PROGRAM PRG_PING_DMX
  VAR
    udiPingTime : UDINT;
    udiDMXnodeReachable : UDINT;
    udiPreviousReachable : UDINT := 16#FFFFFFFF;  (* Last reported result, so the log fires on transitions only. The sentinel differs from every SysSockPing return, so the first pass still logs. *)
    sBrokerHost : STRING;  (* The broker's host without its port. GVL_MQTT.broker carries host:port and SysSockPing wants the host on its own, so it is split here rather than duplicated as a second constant that would drift. Assumes an address of the form ip:port, which is what GVL_MQTT.broker has always held. *)
    iColon : INT;
    udiBrokerPingTime : UDINT;
    udiBrokerReachable : UDINT;
    bPreviousBrokerReachable : BOOL := FALSE;  (* Last logged verdict, so the log fires on transitions only. Deliberately initialised FALSE where bBrokerReachable starts TRUE, so the first verdict is logged whichever way it goes. *)
    uiBrokerPingFails : UINT;  (* Consecutive failed broker pings. One lost ICMP packet must not turn a cabinet LED red, and SysSockPing returns codes that are neither 0 nor 5 - the DMX ping above has always ignored those rather than acting on them. Counting instead of enumerating return codes means an unknown code is treated as a failure without a single one of them being able to flip the light. *)
  END_VAR
  VAR CONSTANT
    cuiBrokerPingFailsForRed : UINT := 2;  (* Failed pings in a row before the broker counts as unreachable. Two, against a 10 s task, means U1 goes red within about 20 s of the cable coming out and green again within 10 s of it going back in. Lower the Ping task period if that is not quick enough; do not lower this to one. *)
  END_VAR

                    (* Ping the DMX artNet node *)
udiDMXnodeReachable := SysSockPing(szIPAddress:=GVL_DMX.IP, ulTimeout:=100, pulReplyTime:= ADR(udiPingTime));

IF udiDMXnodeReachable = 0 THEN
    PFC.SetLed(which:=PFC.LED.U3, how:=PFC.LedState.STATIC_GRN);
	IF udiDMXnodeReachable <> udiPreviousReachable THEN
		GVL_MQTT.PLC_Device.SendLogMessage('DMX ping OK');
	END_IF
ELSIF udiDMXnodeReachable = 5 THEN
     PFC.SetLed(which:=PFC.LED.U3, how:=PFC.LedState.BLINK_RED);
	IF udiDMXnodeReachable <> udiPreviousReachable THEN
		GVL_MQTT.PLC_Device.SendLogMessage('DMX ping Error');
	END_IF
END_IF

udiPreviousReachable := udiDMXnodeReachable;

(* Ping the MQTT broker as well, because U1 needs something the MQTT client cannot
   tell it. MQTT_CONNECTED does not notice a pulled network cable: a TCP socket with
   nothing to report stays open until a retransmit finally gives up, which is minutes
   rather than seconds, so the client goes on believing it has a session. Verified on
   the bench - LAN cable out, MQTT_CONNECTED still TRUE, U1 still green. ICMP notices
   in one task cycle, and the debounce below spends one more, so U1 turns red within
   about 20 s of the cable coming out and green within 10 s of it going back in.

   PRG_MQTT owns the LED; this only reports what it found. *)
iColon := FIND(GVL_MQTT.broker, ':');
IF iColon > 1 THEN
	sBrokerHost := LEFT(GVL_MQTT.broker, iColon - 1);
ELSE
	(* No port in the address, so it is already just the host. FIND returns 0 when
	   it matches nothing, which this also covers. *)
	sBrokerHost := GVL_MQTT.broker;
END_IF

udiBrokerReachable := SysSockPing(szIPAddress := sBrokerHost, ulTimeout := 100,
	pulReplyTime := ADR(udiBrokerPingTime));

(* Debounced, because one lost packet is not an outage. A success clears the count
   immediately, so recovery is as fast as the task; failures have to stack up. *)
IF udiBrokerReachable = 0 THEN
	uiBrokerPingFails := 0;
ELSIF uiBrokerPingFails < cuiBrokerPingFailsForRed THEN
	uiBrokerPingFails := uiBrokerPingFails + 1;
END_IF

GVL_MQTT.bBrokerReachable := (uiBrokerPingFails < cuiBrokerPingFailsForRed);

(* Log the debounced verdict, not the raw return code - otherwise a run of odd
   codes would log on every one of them. *)
IF GVL_MQTT.bBrokerReachable <> bPreviousBrokerReachable THEN
	IF GVL_MQTT.bBrokerReachable THEN
		GVL_MQTT.PLC_Device.SendLogMessage('MQTT broker ping OK');
	ELSE
		(* This one cannot be delivered while the broker is away; it queues and
		   arrives on reconnect, which is what makes the outage visible after the
		   fact rather than not at all. *)
		GVL_MQTT.PLC_Device.SendLogMessage('MQTT broker ping Error');
	END_IF
	bPreviousBrokerReachable := GVL_MQTT.bBrokerReachable;
END_IF

                  
END_PROGRAM

PROGRAM PRG_DALI_VERIFY
  VAR
    Ballast : WagoAppDALI.typBallast := (bAddress := 0, xIsGroup := FALSE, bPortDALI := 1);  (* A ballast on the first 753-647 of this device, short address 0. The values are arbitrary: nothing here is downloaded. What matters is that every type and every call in the DALI chain is compiled on every build. *)
    fbDaliMaster : WagoAppDALI.FbDaliMaster;  (* The master, and the block under test. *)
    fbDimmer : FB_OUTPUT_DIMMER_DALI_MQTT;
  END_VAR

                    // Run the master before anything else, bound to the 753-647 on this device's own
// K-bus. This binding is the whole point of the second controller: I_Port wants a
// WagoTypesModule_753_647.I_Port_753_647, which only WAGO's device description
// creates, and that description does not fit the G1 lab device's bus.
fbDaliMaster(
	bPortDALI := 1,
	I_Port := IoConfig_Globals.DALI_753_647);

// The block under test. No InitMqtt and no InitMqttDiscovery: this application
// never runs, and calling them would only invent a Home Assistant entity for a
// controller that does not exist.
fbDimmer(
	BALLAST := Ballast,
	TOGGLE := FALSE,
	P_LONG := FALSE);

                  
END_PROGRAM

CONFIGURATION Wago_PFC200_G1_Lab
  RESOURCE HomeAutomation ON PLC
    {attribute 'qualified_only'}
    VAR_GLOBAL CONSTANT  (* GVL_MQTT *)
      MQTT_TOPIC_LEN : INT := 160;  (* Widths for topics and topic fragments. These used to be spelled out at five different values for the same conceptual string, and IEC string assignment and CONCAT both truncate without any error - so every mismatch was a silent failure point. The tightest real chain: a 28-character prefix like 'Devices/PLC/Lab/Out/Dimmers/' plus a 40-character instance name plus '/OUT' already reached the old STRING(100) limit, after which Home Assistant sees a truncated state topic and the entity goes quietly unavailable. *)
      MQTT_SUFFIX_LEN : INT := 64;
      clientID : STRING := 'PLC-Lab';  (* Broker setup *)
      broker : STRING := '10.101.1.11:1883';
      fbMqttPublishQueue : FB_MQTT_PUBLISH_QUEUE;  (* use the below for username password authentication to broker broker :STRING:='user:password@192.168.1.36:1883'; Shared Variables for MQTT publish communication *)
      collector_FB_OUTPUT_SWITCH_MQTT : MQTT.CallbackCollector;  (* Shared Variables for MQTT subscribe communication *)
      collector_FB_OUTPUT_COVER_MQTT : MQTT.CallbackCollector;
      collector_FB_DIMMER_MQTT : MQTT.CallbackCollector;
      collector_FB_RS485_MQTT : MQTT.CallbackCollector;
      collector_FB_HVAC_MQTT : MQTT.CallbackCollector;
      MQTT_QOS_EXACTLY_ONCE : MQTT.QoS := MQTT.QoS.ExactlyOnce;  (* QOS Constants *)
      MqttMain : STRING(16) := 'Devices/';  (* Topics *)
      MqttType : STRING(16) := 'PLC/';
      MqttDevice : STRING(16) := 'Lab/';
      MqttBaseTopic : STRING(GVL_MQTT.MQTT_TOPIC_LEN) := 'CONCAT(CONCAT(MqttMain, MqttType), MqttDevice)';  (* e.g. Devices/PLC/House *)
      MqttDiagnosticTopic : STRING(GVL_MQTT.MQTT_TOPIC_LEN) := 'CONCAT(MqttBaseTopic, 'diagnostic')';
      MqttAvailabilityTopic : STRING(GVL_MQTT.MQTT_TOPIC_LEN) := 'CONCAT(MqttBaseTopic, 'availability')';
      MqttAvailabilityOnlinePayload : STRING(20) := 'online';
      MqttAvailabilityOfflinePayload : STRING(20) := 'offline';
      MQTTAvailabilityHartbeatTime : TIME := TIME#5s0ms;
      MqttHADiscoveryPrefix : STRING(16) := 'homeassistant/';
      PLC_Device : FB_PLC_MQTT_DISCOVERY_DEVICE;  (* HOME ASSISTANT DISCOVERY VIA MQTT *)
      OWD_MULTISENSOR_01 : FB_1WIRE_MQTT_DISCOVERY_DEVICE;
      MqttPushbuttonPrefix : STRING(GVL_MQTT.MQTT_TOPIC_LEN) := 'CONCAT(MqttBaseTopic, 'Out/DigitalInputs/Pushbuttons/')';  (* FB Topics *)
      MqttPubSwitchPrefix : STRING(GVL_MQTT.MQTT_TOPIC_LEN) := 'CONCAT(MqttBaseTopic, 'Out/DigitalOutputs/')';
      MqttSubSwitchPrefix : STRING(GVL_MQTT.MQTT_TOPIC_LEN) := 'CONCAT(MqttBaseTopic, 'In/DigitalOutputs/')';
      MqttPubCoverPrefix : STRING(GVL_MQTT.MQTT_TOPIC_LEN) := 'CONCAT(MqttBaseTopic, 'Out/Covers/')';
      MqttSubCoverPrefix : STRING(GVL_MQTT.MQTT_TOPIC_LEN) := 'CONCAT(MqttBaseTopic, 'In/Covers/')';
      MqttPubDimmerPrefix : STRING(GVL_MQTT.MQTT_TOPIC_LEN) := 'CONCAT(MqttBaseTopic, 'Out/Dimmers/')';
      MqttSubDimmerPrefix : STRING(GVL_MQTT.MQTT_TOPIC_LEN) := 'CONCAT(MqttBaseTopic, 'In/Dimmers/')';
      MqttPubRS485Prefix : STRING(GVL_MQTT.MQTT_TOPIC_LEN) := 'CONCAT(MqttBaseTopic, 'Out/RS485/')';
      MqttSubRS485Prefix : STRING(GVL_MQTT.MQTT_TOPIC_LEN) := 'CONCAT(MqttBaseTopic, 'In/RS485/')';
      MqttPubHVACPrefix : STRING(GVL_MQTT.MQTT_TOPIC_LEN) := 'CONCAT(MqttBaseTopic, 'Out/HVAC/')';
      MqttPubAnalogInputPrefix : STRING(GVL_MQTT.MQTT_TOPIC_LEN) := 'CONCAT(MqttBaseTopic, 'Out/AnalogInputs/')';  (* On-board analog inputs: an RTD channel on a 750-463, and anything else measured by the PLC itself rather than over a bus. Publish only - there is nothing to command on an input. *)
      MqttSubHVACPrefix : STRING(GVL_MQTT.MQTT_TOPIC_LEN) := 'CONCAT(MqttBaseTopic, 'In/HVAC/')';
      MqttSubSwitchTopic : STRING(GVL_MQTT.MQTT_TOPIC_LEN) := 'CONCAT(MqttSubSwitchPrefix, '+')';  (* Wildcard subscriptions *)
      MqttSubCoverTopic : STRING(GVL_MQTT.MQTT_TOPIC_LEN) := 'CONCAT(MqttSubCoverPrefix, '#')';  (* '#', not '+': the position command topic sits one level below the cover's own topic - .../In/Covers/FB_X/POSITION - and a single-level wildcard would not deliver it. The older cover block's topics still match. *)
      MqttSubDimmerTopic : STRING(GVL_MQTT.MQTT_TOPIC_LEN) := 'CONCAT(MqttSubDimmerPrefix, '#')';
      MqttSubRS485Topic : STRING(GVL_MQTT.MQTT_TOPIC_LEN) := 'CONCAT(MqttSubRS485Prefix, '#')';
      MqttSubHVACTopic : STRING(GVL_MQTT.MQTT_TOPIC_LEN) := 'CONCAT(MqttSubHVACPrefix, '#')';
      bBrokerReachable : BOOL := TRUE;  (* TRUE while the broker host answers an ICMP ping. Written by PRG_PING_DMX, read by PRG_MQTT, which ANDs it with the client's own MQTT_CONNECTED before deciding what U1 shows. It is not redundant. MQTT_CONNECTED does not notice a pulled network cable: TCP has nothing to report until a retransmit gives up, so the client can hold a dead socket open for minutes. Measured on the bench - cable out, U1 stayed green. ICMP notices within one cycle of the Ping task. Starts TRUE so it means 'not known to be unreachable': until the Ping task has an opinion, U1 follows MQTT_CONNECTED alone rather than blinking red through a healthy startup. *)
      MQTT_LANE_MAIN : INT := 0;
      MQTT_LANE_RS485 : INT := 1;
      MQTT_LANE_HVAC : INT := 2;
      tMqttReconnectRestMin : TIME := TIME#1s0ms;  (* Reconnect pacing, read by PRG_MQTT. They live here rather than in an FB_init argument or an initialiser because both of those are stored outside the declaration text, where a scripted edit cannot reach them. First pause after a session drops, and the ceiling the pause doubles towards. One second is short enough that an ordinary reconnect is not noticeably slower; a minute is the worst the broker ever sees. *)
      tMqttReconnectRestMax : TIME := TIME#1m0s0ms;
      tMqttSessionStable : TIME := TIME#30s0ms;  (* How long a session has to last before it counts as a real one. Long enough that a session which dies on arrival cannot clear the backoff, short enough that a healthy reconnect clears it well before the next heartbeat. *)
      tMqttStall : TIME := TIME#5m0s0ms;  (* No stable session for this long is a stall, not bad luck: the client stops trying for tMqttStallCoolDown and then starts again. *)
      tMqttStallCoolDown : TIME := TIME#1m0s0ms;
    END_VAR
    {attribute 'qualified_only'}
    VAR_GLOBAL  (* GVL_DMX *)
      IP : STRING := '10.1.1.4';  (* unicast: 10.1.1.4 multicast: 10.1.1.255 broadcast: 255.255.255.255 *)
      DMX : oscat_network.NETWORK_BUFFER_SHORT;
    END_VAR
    {attribute 'qualified_only'}
    VAR_GLOBAL  (* GVL_RS485 *)
      FB_RS485_EASTRON_SDM220_1 : FB_RS485_EASTRON_SDM220_MQTT := (FriendlyName := 'Lab PLC SDM220 energy meter');  (* RS485 *)
      FB_RS485_DUCO_DUCOBOX_HOME : FB_RS485_DUCO_DUCOBOX_FOCUS_MQTT;
      FB_RS485_1WIRE_MULTISENSOR_01 : FB_RS485_ESERA_OWD_MQTT;
      FB_RS485_EASTRON_SDM630_1 : FB_RS485_EASTRON_SDM630_MQTT := (FriendlyName := 'Lab PLC energy meter');  (* Self-wiring: FriendlyName is what turns the MQTT and discovery wiring on, so this needs no Init call in RS485_INIT - only registration on the bus. *)
      FB_RS485_EASTRON_SDM_POWER_1 : FB_RS485_EASTRON_SDM_POWER_MQTT := (FriendlyName := 'Lab PLC SDM power meter');  (* Registered on the bus and pointed at the SAME meter as FB_RS485_EASTRON_SDM220_1 above (Modbus address 1), declared as an SDM220. That is deliberate on two counts. It is the only call site this block has, and an unreferenced POU is never compiled - without an instance somewhere in the application a broken edit to it would pass verify with a clean build. And because both blocks decode active power out of the same register (30013), the two publish the same number continuously: a persistent difference between .../FB_RS485_EASTRON_SDM_POWER_1/ACTP and .../FB_RS485_EASTRON_SDM220_1/ACTP means one of them has stopped decoding correctly. There is no SDM120 or SDM630 here, so this is the only way the block is exercised at all. *)
      FB_RS485_SEN0492_1 : FB_RS485_DFROBOT_SEN0492_MQTT := (FriendlyName := 'Lab PLC rangefinder');  (* DFRobot SEN0492 laser rangefinder, 4 cm to 4 m over RS485. Left at its factory slave address 16#50, which collides with nothing on this bus - the Eastron meters sit at 1 and 4. Only the baud rate has to be changed, and the sensor asks for that itself at startup - see its GetCommissioning, and FB_RS485_COMMISSIONER which acts on it. *)
      RS485_COMMISSION_ON_BOOT : BOOL := TRUE;  (* Run commissioning on every startup: before the bus controller is allowed to poll anything, every registered device is asked whether it needs something written into it first - see FB_RS485_COMMISSIONER. A device that answers no, which is nearly all of them, costs one method call. It is worth doing every boot rather than once, because it also repairs a device somebody has factory-reset. Set FALSE to skip it entirely: the sequence holds the bus controller off while it runs, so on a bus where nothing needs commissioning this saves nothing but is the switch to reach for if a sweep ever misbehaves. *)
    END_VAR
    TASK HvacTask(INTERVAL := T#50ms, PRIORITY := 8);
    TASK MainTask(INTERVAL := T#50ms, PRIORITY := 4);
    TASK MqttCommunication(INTERVAL := T#20ms, PRIORITY := 5);
    TASK Ping(INTERVAL := T#10000ms, PRIORITY := 31);
    TASK RS485(INTERVAL := T#50ms, PRIORITY := 15);
    PROGRAM PRG_HVAC WITH HvacTask : PRG_HVAC;
    PROGRAM PRG_MAIN WITH MainTask : PRG_MAIN;
    PROGRAM PRG_MQTT WITH MqttCommunication : PRG_MQTT;
    PROGRAM PRG_DMX_SEND WITH MqttCommunication : PRG_DMX_SEND;
    PROGRAM PRG_PING_DMX WITH Ping : PRG_PING_DMX;
    PROGRAM PRG_RS485 WITH RS485 : PRG_RS485;
  END_RESOURCE
END_CONFIGURATION

CONFIGURATION Pfc200Bus
END_CONFIGURATION

CONFIGURATION _75x_440
END_CONFIGURATION

CONFIGURATION _75x_540
END_CONFIGURATION

CONFIGURATION _75x_540_1
END_CONFIGURATION

CONFIGURATION _75x_467
END_CONFIGURATION

CONFIGURATION _75x_550
END_CONFIGURATION

CONFIGURATION Wago_PFC200_G2_Virtual
  RESOURCE Application ON PLC
    {attribute 'qualified_only'}
    VAR_GLOBAL CONSTANT  (* GVL_MQTT *)
      MQTT_TOPIC_LEN : INT := 160;  (* The only two members FB_MQTT_BASE and FB_MQTT_PUBLISH_QUEUE read, and so the only two this application needs: it exists to compile the DALI chain, not to speak MQTT. The real GVL_MQTT lives in Wago_PFC200_G1_Lab's application, and a GVL cannot be shared between applications. If these drift from the real ones nothing breaks here - they only size strings, and this application is never downloaded. *)
      MQTT_SUFFIX_LEN : INT := 64;
      MQTT_LANE_MAIN : INT := 0;
      MQTT_LANE_RS485 : INT := 1;
      MQTT_LANE_HVAC : INT := 2;
    END_VAR
    TASK DaliVerify(INTERVAL := T#200ms, PRIORITY := 15);
    PROGRAM PRG_DALI_VERIFY WITH DaliVerify : PRG_DALI_VERIFY;
  END_RESOURCE
END_CONFIGURATION

CONFIGURATION Kbus
END_CONFIGURATION

CONFIGURATION DALI_753_647
END_CONFIGURATION

CONFIGURATION Serial
END_CONFIGURATION

CONFIGURATION COM1
END_CONFIGURATION
